FUNCTION_BLOCK FB_Scheduler_F53
      VAR_INPUT
          currH : WORD;
          currM : WORD;
          currD : WORD;
      END_VAR
      VAR_IN_OUT
          FB_Bacnet : FB_BACnet_DAIKIN_MasterStation_III_No_10;
      END_VAR
      VAR
          i : INT;
          bUnitTriggered : BOOL := FALSE; // New flag to track execution
          prevMinute : WORD := 0;        // New variable to track the previous minute
      END_VAR
      VAR PERSISTENT
          //scheduler var
          bEnSchedF53_ : BOOL := FALSE;
          wSchedWDHourStartF53_ : WORD; 
          wSchedWDMinStartF53_ : WORD; 
          wSchedWEHourStartF53_ : WORD; 
          wSchedWEMinStartF53_ : WORD;
          wSchedWDHourEndF53_ : WORD;
          wSchedWDMinEndF53_ : WORD;
          wSchedWEHourEndF53_ : WORD;
          wSchedWEMinEndF53_ : WORD;
          //unit var
          bUnitF53_ : ARRAY [1..25] OF BOOL;
      END_VAR


// Reset trigger flag at minute change or at the exact scheduled time
IF currM <> prevMinute OR 
   (currH = wSchedWDHourStartF53_ AND currM = wSchedWDMinStartF53_) OR 
   (currH = wSchedWDHourEndF53_ AND currM = wSchedWDMinEndF53_) THEN
    bUnitTriggered := FALSE;
    prevMinute := currM;
END_IF

// Unit Schedule Enable
IF bEnSchedF53_ THEN
    // Weekday schedule
    IF currD >= 1 AND currD <= 5 THEN
        IF (wSchedWDHourStartF53_ <> wSchedWDHourEndF53_ OR wSchedWDMinStartF53_ <> wSchedWDMinEndF53_) THEN
            // Schedule Unit ON
            IF wSchedWDHourStartF53_ = currH AND wSchedWDMinStartF53_ = currM AND NOT bUnitTriggered THEN
                bUnitTriggered := TRUE;
                FOR i := 1 TO 25 DO
                    //send command unit ON
                    IF bUnitF53_[i] = TRUE THEN 
                        CASE i OF
                            1: 
                                FB_Bacnet.StartStopCommand_192.bEnWrite := TRUE;
                                FB_Bacnet.StartStopCommand_192.bVal := TRUE;
                            2: 
                                FB_Bacnet.StartStopCommand_193.bEnWrite := TRUE;
                                FB_Bacnet.StartStopCommand_193.bVal := TRUE;
                            3: 
                                FB_Bacnet.StartStopCommand_194.bEnWrite := TRUE;
                                FB_Bacnet.StartStopCommand_194.bVal := TRUE;
                            4: 
                                FB_Bacnet.StartStopCommand_195.bEnWrite := TRUE;
                                FB_Bacnet.StartStopCommand_195.bVal := TRUE;
                            5: 
                                FB_Bacnet.StartStopCommand_196.bEnWrite := TRUE;
                                FB_Bacnet.StartStopCommand_196.bVal := TRUE;
                            6: 
                                FB_Bacnet.StartStopCommand_197.bEnWrite := TRUE;
                                FB_Bacnet.StartStopCommand_197.bVal := TRUE;
                            7: 
                                FB_Bacnet.StartStopCommand_198.bEnWrite := TRUE;
                                FB_Bacnet.StartStopCommand_198.bVal := TRUE;
                            8: 
                                FB_Bacnet.StartStopCommand_199.bEnWrite := TRUE;
                                FB_Bacnet.StartStopCommand_199.bVal := TRUE;
                            9: 
                                //FB_Bacnet.StartStopCommand_200.bEnWrite := TRUE;
                                //FB_Bacnet.StartStopCommand_200.bVal := TRUE;
                            10: 
                                FB_Bacnet.StartStopCommand_201.bEnWrite := TRUE;
                                FB_Bacnet.StartStopCommand_201.bVal := TRUE;
                            11: 
                                FB_Bacnet.StartStopCommand_202.bEnWrite := TRUE;
                                FB_Bacnet.StartStopCommand_202.bVal := TRUE;
                            12: 
                                FB_Bacnet.StartStopCommand_203.bEnWrite := TRUE;
                                FB_Bacnet.StartStopCommand_203.bVal := TRUE;
                            13: 
                                FB_Bacnet.StartStopCommand_204.bEnWrite := TRUE;
                                FB_Bacnet.StartStopCommand_204.bVal := TRUE;
                            14: 
                                FB_Bacnet.StartStopCommand_205.bEnWrite := TRUE;
                                FB_Bacnet.StartStopCommand_205.bVal := TRUE;
                            15: 
                                FB_Bacnet.StartStopCommand_206.bEnWrite := TRUE;
                                FB_Bacnet.StartStopCommand_206.bVal := TRUE;
                            16: 
                                FB_Bacnet.StartStopCommand_207.bEnWrite := TRUE;
                                FB_Bacnet.StartStopCommand_207.bVal := TRUE;
                            17: 
                                FB_Bacnet.StartStopCommand_208.bEnWrite := TRUE;
                                FB_Bacnet.StartStopCommand_208.bVal := TRUE;
                            18: 
                                FB_Bacnet.StartStopCommand_209.bEnWrite := TRUE;
                                FB_Bacnet.StartStopCommand_209.bVal := TRUE;
                            19: 
                                FB_Bacnet.StartStopCommand_210.bEnWrite := TRUE;
                                FB_Bacnet.StartStopCommand_210.bVal := TRUE;
                            20: 
                                FB_Bacnet.StartStopCommand_211.bEnWrite := TRUE;
                                FB_Bacnet.StartStopCommand_211.bVal := TRUE;
                            21: 
                                FB_Bacnet.StartStopCommand_212.bEnWrite := TRUE;
                                FB_Bacnet.StartStopCommand_212.bVal := TRUE;
                            22: 
                                FB_Bacnet.StartStopCommand_213.bEnWrite := TRUE;
                                FB_Bacnet.StartStopCommand_213.bVal := TRUE;
                            23: 
                                FB_Bacnet.StartStopCommand_242.bEnWrite := TRUE;
                                FB_Bacnet.StartStopCommand_242.bVal := TRUE;
                            24: 
                                FB_Bacnet.StartStopCommand_243.bEnWrite := TRUE;
                                FB_Bacnet.StartStopCommand_243.bVal := TRUE;
                            25: 
                                FB_Bacnet.StartStopCommand_237.bEnWrite := TRUE;
                                FB_Bacnet.StartStopCommand_237.bVal := TRUE;
                        END_CASE
                    END_IF
                END_FOR
            END_IF
            // Schedule Unit OFF
            IF wSchedWDHourEndF53_ = currH AND wSchedWDMinEndF53_ = currM AND NOT bUnitTriggered THEN
                bUnitTriggered := TRUE;
                FOR i := 1 TO 25 DO
                    //send command unit OFF
                    IF bUnitF53_[i] = TRUE THEN 
                        CASE i OF
                            1: 
                                FB_Bacnet.StartStopCommand_192.bEnWrite := TRUE;
                                FB_Bacnet.StartStopCommand_192.bVal := FALSE;
                            2: 
                                FB_Bacnet.StartStopCommand_193.bEnWrite := TRUE;
                                FB_Bacnet.StartStopCommand_193.bVal := FALSE;
                            3: 
                                FB_Bacnet.StartStopCommand_194.bEnWrite := TRUE;
                                FB_Bacnet.StartStopCommand_194.bVal := FALSE;
                            4: 
                                FB_Bacnet.StartStopCommand_195.bEnWrite := TRUE;
                                FB_Bacnet.StartStopCommand_195.bVal := FALSE;
                            5: 
                                FB_Bacnet.StartStopCommand_196.bEnWrite := TRUE;
                                FB_Bacnet.StartStopCommand_196.bVal := FALSE;
                            6: 
                                FB_Bacnet.StartStopCommand_197.bEnWrite := TRUE;
                                FB_Bacnet.StartStopCommand_197.bVal := FALSE;
                            7: 
                                FB_Bacnet.StartStopCommand_198.bEnWrite := TRUE;
                                FB_Bacnet.StartStopCommand_198.bVal := FALSE;
                            8: 
                                FB_Bacnet.StartStopCommand_199.bEnWrite := TRUE;
                                FB_Bacnet.StartStopCommand_199.bVal := FALSE;
                            9: 
                                //FB_Bacnet.StartStopCommand_200.bEnWrite := TRUE;
                                //FB_Bacnet.StartStopCommand_200.bVal := FALSE;
                            10: 
                                FB_Bacnet.StartStopCommand_201.bEnWrite := TRUE;
                                FB_Bacnet.StartStopCommand_201.bVal := FALSE;
                            11: 
                                FB_Bacnet.StartStopCommand_202.bEnWrite := TRUE;
                                FB_Bacnet.StartStopCommand_202.bVal := FALSE;
                            12: 
                                FB_Bacnet.StartStopCommand_203.bEnWrite := TRUE;
                                FB_Bacnet.StartStopCommand_203.bVal := FALSE;
                            13: 
                                FB_Bacnet.StartStopCommand_204.bEnWrite := TRUE;
                                FB_Bacnet.StartStopCommand_204.bVal := FALSE;
                            14: 
                                FB_Bacnet.StartStopCommand_205.bEnWrite := TRUE;
                                FB_Bacnet.StartStopCommand_205.bVal := FALSE;
                            15: 
                                FB_Bacnet.StartStopCommand_206.bEnWrite := TRUE;
                                FB_Bacnet.StartStopCommand_206.bVal := FALSE;
                            16: 
                                FB_Bacnet.StartStopCommand_207.bEnWrite := TRUE;
                                FB_Bacnet.StartStopCommand_207.bVal := FALSE;
                            17: 
                                FB_Bacnet.StartStopCommand_208.bEnWrite := TRUE;
                                FB_Bacnet.StartStopCommand_208.bVal := FALSE;
                            18: 
                                FB_Bacnet.StartStopCommand_209.bEnWrite := TRUE;
                                FB_Bacnet.StartStopCommand_209.bVal := FALSE;
                            19: 
                                FB_Bacnet.StartStopCommand_210.bEnWrite := TRUE;
                                FB_Bacnet.StartStopCommand_210.bVal := FALSE;
                            20: 
                                FB_Bacnet.StartStopCommand_211.bEnWrite := TRUE;
                                FB_Bacnet.StartStopCommand_211.bVal := FALSE;
                            21: 
                                FB_Bacnet.StartStopCommand_212.bEnWrite := TRUE;
                                FB_Bacnet.StartStopCommand_212.bVal := FALSE;
                            22: 
                                FB_Bacnet.StartStopCommand_213.bEnWrite := TRUE;
                                FB_Bacnet.StartStopCommand_213.bVal := FALSE;
                            23: 
                                FB_Bacnet.StartStopCommand_242.bEnWrite := TRUE;
                                FB_Bacnet.StartStopCommand_242.bVal := FALSE;
                            24: 
                                FB_Bacnet.StartStopCommand_243.bEnWrite := TRUE;
                                FB_Bacnet.StartStopCommand_243.bVal := FALSE;
                            25: 
                                FB_Bacnet.StartStopCommand_237.bEnWrite := TRUE;
                                FB_Bacnet.StartStopCommand_237.bVal := FALSE;
                        END_CASE
                    END_IF
                END_FOR
            END_IF
        END_IF
    END_IF

    // Weekend schedule
    IF currD = 0 OR currD = 6 THEN
        IF (wSchedWEHourStartF53_ <> wSchedWEHourEndF53_ OR wSchedWEMinStartF53_ <> wSchedWEMinEndF53_) THEN
            // Schedule Unit ON
            IF wSchedWEHourStartF53_ = currH AND wSchedWEMinStartF53_ = currM AND NOT bUnitTriggered THEN
                bUnitTriggered := TRUE;
                FOR i := 1 TO 25 DO
                    //send command unit ON
                    IF bUnitF53_[i] = TRUE THEN 
                        CASE i OF
                            1: 
                                FB_Bacnet.StartStopCommand_192.bEnWrite := TRUE;
                                FB_Bacnet.StartStopCommand_192.bVal := TRUE;
                            2: 
                                FB_Bacnet.StartStopCommand_193.bEnWrite := TRUE;
                                FB_Bacnet.StartStopCommand_193.bVal := TRUE;
                            3: 
                                FB_Bacnet.StartStopCommand_194.bEnWrite := TRUE;
                                FB_Bacnet.StartStopCommand_194.bVal := TRUE;
                            4: 
                                FB_Bacnet.StartStopCommand_195.bEnWrite := TRUE;
                                FB_Bacnet.StartStopCommand_195.bVal := TRUE;
                            5: 
                                FB_Bacnet.StartStopCommand_196.bEnWrite := TRUE;
                                FB_Bacnet.StartStopCommand_196.bVal := TRUE;
                            6: 
                                FB_Bacnet.StartStopCommand_197.bEnWrite := TRUE;
                                FB_Bacnet.StartStopCommand_197.bVal := TRUE;
                            7: 
                                FB_Bacnet.StartStopCommand_198.bEnWrite := TRUE;
                                FB_Bacnet.StartStopCommand_198.bVal := TRUE;
                            8: 
                                FB_Bacnet.StartStopCommand_199.bEnWrite := TRUE;
                                FB_Bacnet.StartStopCommand_199.bVal := TRUE;
                            9: 
                                //FB_Bacnet.StartStopCommand_200.bEnWrite := TRUE;
                                //FB_Bacnet.StartStopCommand_200.bVal := TRUE;
                            10: 
                                FB_Bacnet.StartStopCommand_201.bEnWrite := TRUE;
                                FB_Bacnet.StartStopCommand_201.bVal := TRUE;
                            11: 
                                FB_Bacnet.StartStopCommand_202.bEnWrite := TRUE;
                                FB_Bacnet.StartStopCommand_202.bVal := TRUE;
                            12: 
                                FB_Bacnet.StartStopCommand_203.bEnWrite := TRUE;
                                FB_Bacnet.StartStopCommand_203.bVal := TRUE;
                            13: 
                                FB_Bacnet.StartStopCommand_204.bEnWrite := TRUE;
                                FB_Bacnet.StartStopCommand_204.bVal := TRUE;
                            14: 
                                FB_Bacnet.StartStopCommand_205.bEnWrite := TRUE;
                                FB_Bacnet.StartStopCommand_205.bVal := TRUE;
                            15: 
                                FB_Bacnet.StartStopCommand_206.bEnWrite := TRUE;
                                FB_Bacnet.StartStopCommand_206.bVal := TRUE;
                            16: 
                                FB_Bacnet.StartStopCommand_207.bEnWrite := TRUE;
                                FB_Bacnet.StartStopCommand_207.bVal := TRUE;
                            17: 
                                FB_Bacnet.StartStopCommand_208.bEnWrite := TRUE;
                                FB_Bacnet.StartStopCommand_208.bVal := TRUE;
                            18: 
                                FB_Bacnet.StartStopCommand_209.bEnWrite := TRUE;
                                FB_Bacnet.StartStopCommand_209.bVal := TRUE;
                            19: 
                                FB_Bacnet.StartStopCommand_210.bEnWrite := TRUE;
                                FB_Bacnet.StartStopCommand_210.bVal := TRUE;
                            20: 
                                FB_Bacnet.StartStopCommand_211.bEnWrite := TRUE;
                                FB_Bacnet.StartStopCommand_211.bVal := TRUE;
                            21: 
                                FB_Bacnet.StartStopCommand_212.bEnWrite := TRUE;
                                FB_Bacnet.StartStopCommand_212.bVal := TRUE;
                            22: 
                                FB_Bacnet.StartStopCommand_213.bEnWrite := TRUE;
                                FB_Bacnet.StartStopCommand_213.bVal := TRUE;
                            23: 
                                FB_Bacnet.StartStopCommand_242.bEnWrite := TRUE;
                                FB_Bacnet.StartStopCommand_242.bVal := TRUE;
                            24: 
                                FB_Bacnet.StartStopCommand_243.bEnWrite := TRUE;
                                FB_Bacnet.StartStopCommand_243.bVal := TRUE;
                            25: 
                                FB_Bacnet.StartStopCommand_237.bEnWrite := TRUE;
                                FB_Bacnet.StartStopCommand_237.bVal := TRUE;
                        END_CASE
                    END_IF
                END_FOR        
            END_IF
            // Schedule Unit OFF
            IF wSchedWEHourEndF53_ = currH AND wSchedWEMinEndF53_ = currM AND NOT bUnitTriggered THEN
                bUnitTriggered := TRUE;
                FOR i := 1 TO 25 DO
                    //send command unit OFF
                    IF bUnitF53_[i] = TRUE THEN 
                        CASE i OF
                            1: 
                                FB_Bacnet.StartStopCommand_192.bEnWrite := TRUE;
                                FB_Bacnet.StartStopCommand_192.bVal := FALSE;
                            2: 
                                FB_Bacnet.StartStopCommand_193.bEnWrite := TRUE;
                                FB_Bacnet.StartStopCommand_193.bVal := FALSE;
                            3: 
                                FB_Bacnet.StartStopCommand_194.bEnWrite := TRUE;
                                FB_Bacnet.StartStopCommand_194.bVal := FALSE;
                            4: 
                                FB_Bacnet.StartStopCommand_195.bEnWrite := TRUE;
                                FB_Bacnet.StartStopCommand_195.bVal := FALSE;
                            5: 
                                FB_Bacnet.StartStopCommand_196.bEnWrite := TRUE;
                                FB_Bacnet.StartStopCommand_196.bVal := FALSE;
                            6: 
                                FB_Bacnet.StartStopCommand_197.bEnWrite := TRUE;
                                FB_Bacnet.StartStopCommand_197.bVal := FALSE;
                            7: 
                                FB_Bacnet.StartStopCommand_198.bEnWrite := TRUE;
                                FB_Bacnet.StartStopCommand_198.bVal := FALSE;
                            8: 
                                FB_Bacnet.StartStopCommand_199.bEnWrite := TRUE;
                                FB_Bacnet.StartStopCommand_199.bVal := FALSE;
                            9: 
                                //FB_Bacnet.StartStopCommand_200.bEnWrite := TRUE;
                                //FB_Bacnet.StartStopCommand_200.bVal := FALSE;
                            10: 
                                FB_Bacnet.StartStopCommand_201.bEnWrite := TRUE;
                                FB_Bacnet.StartStopCommand_201.bVal := FALSE;
                            11: 
                                FB_Bacnet.StartStopCommand_202.bEnWrite := TRUE;
                                FB_Bacnet.StartStopCommand_202.bVal := FALSE;
                            12: 
                                FB_Bacnet.StartStopCommand_203.bEnWrite := TRUE;
                                FB_Bacnet.StartStopCommand_203.bVal := FALSE;
                            13: 
                                FB_Bacnet.StartStopCommand_204.bEnWrite := TRUE;
                                FB_Bacnet.StartStopCommand_204.bVal := FALSE;
                            14: 
                                FB_Bacnet.StartStopCommand_205.bEnWrite := TRUE;
                                FB_Bacnet.StartStopCommand_205.bVal := FALSE;
                            15: 
                                FB_Bacnet.StartStopCommand_206.bEnWrite := TRUE;
                                FB_Bacnet.StartStopCommand_206.bVal := FALSE;
                            16: 
                                FB_Bacnet.StartStopCommand_207.bEnWrite := TRUE;
                                FB_Bacnet.StartStopCommand_207.bVal := FALSE;
                            17: 
                                FB_Bacnet.StartStopCommand_208.bEnWrite := TRUE;
                                FB_Bacnet.StartStopCommand_208.bVal := FALSE;
                            18: 
                                FB_Bacnet.StartStopCommand_209.bEnWrite := TRUE;
                                FB_Bacnet.StartStopCommand_209.bVal := FALSE;
                            19: 
                                FB_Bacnet.StartStopCommand_210.bEnWrite := TRUE;
                                FB_Bacnet.StartStopCommand_210.bVal := FALSE;
                            20: 
                                FB_Bacnet.StartStopCommand_211.bEnWrite := TRUE;
                                FB_Bacnet.StartStopCommand_211.bVal := FALSE;
                            21: 
                                FB_Bacnet.StartStopCommand_212.bEnWrite := TRUE;
                                FB_Bacnet.StartStopCommand_212.bVal := FALSE;
                            22: 
                                FB_Bacnet.StartStopCommand_213.bEnWrite := TRUE;
                                FB_Bacnet.StartStopCommand_213.bVal := FALSE;
                            23: 
                                FB_Bacnet.StartStopCommand_242.bEnWrite := TRUE;
                                FB_Bacnet.StartStopCommand_242.bVal := FALSE;
                            24: 
                                FB_Bacnet.StartStopCommand_243.bEnWrite := TRUE;
                                FB_Bacnet.StartStopCommand_243.bVal := FALSE;
                            25: 
                                FB_Bacnet.StartStopCommand_237.bEnWrite := TRUE;
                                FB_Bacnet.StartStopCommand_237.bVal := FALSE;
                        END_CASE
                    END_IF
                END_FOR
            END_IF
        END_IF
    END_IF
END_IF

END_FUNCTION_BLOCK

(* stored: Version 1.1.0.1, ProductVersion 3.1.4024.14
   POU FB_Scheduler_F53: Id {820f1807-65a3-4536-a630-522d2bea77b9}, SpecialFunc None *)
